TYPE ST_HMI_Monitor_OCP : //overcurrent protection
STRUCT
	b_InputMCCBstate			: BOOL;
	b_OutputMCCBstate			: BOOL;
	b_InputOverloadWarning		: BOOL;
	b_InputOverloadAlarm		: BOOL;
	b_OutputOverloadWarning		: BOOL;
	b_OutputOverloadAlarm		: BOOL;
	s_Location					: STRING;
	r_CurrentPeak				: REAL;
	t_PeakDuration				: TIME;	
END_STRUCT
END_TYPE

(* stored: Version 1.1.0.1, ProductVersion 3.1.4026.18
   DUT ST_HMI_Monitor_OCP: Id {82419d34-2980-4dfe-adfc-46343c87ccde} *)
